// TIA Portal V16 export
// export: Created 2024-09-05T17:40:14.0276787Z, ExportSetting WithDefaults, DisplayName Totally Integrated Automation Portal, DisplayVersion V16 Update 6, DisplayName TIA Portal Version Control Interface, DisplayVersion V16 Update 2, DisplayName TIA Portal Openness, DisplayVersion V16 Update 6, DisplayName STEP 7 Professional, DisplayVersion V16 Update 6, DisplayName STEP 7 Safety, DisplayVersion V16, DisplayName WinCC Advanced, DisplayVersion V16 Update 6
TYPE "READER_PRODUCT"
// stored: IsFailsafeCompliant false
   STRUCT
      SIDE_RH : Struct
         POSITION : Int;
         LEN : Int;
         STRING_LABEL : String;
         READER_BYPASS : Bool;
      END_STRUCT;
      SIDE_LH : Struct
         POSITION : Int;
         LEN : Int;
         STRING_LABEL : String;
         READER_BYPASS : Bool;
      END_STRUCT;
      REAR_TUBE : Struct
         POSITION : Int;
         LEN : Int;
         STRING_LABEL : String;
         READER_BYPASS : Bool;
      END_STRUCT;
      FRONT_TUBE : Struct
         POSITION : Int;
         LEN : Int;
         STRING_LABEL : String;
         READER_BYPASS : Bool;
      END_STRUCT;
      NUM_TUBE : Bool;   // 0 = 1 TUBE 1 = 2 TUBES
   END_STRUCT;
END_TYPE
